screen "Automatski" 800x480
   TextField "Text field_2" at 681,0 size 116x23; Text 'Alen Lacković'
   Switch "Switch_1" at 95,185 size 160x80; CaptionText 'Switch'; TextOff 'OFF'; TextOn 'ON'
      ProcessValue <- "Automatsko_upravljanje_Paletizacija"
   TextField "Text field_4" at 95,155 size 121x28; Text 'Paletizacija'
   SymbolicIOField "Symbolic I/O field_1" at 40,317 size 130x50; TextOff '0'; TextOn '1'; TextList "Broj_komada_u_paleti_x-os"
      ProcessValue <- "Automatsko_upravljanje_Broj_komada_palete_x"
   SymbolicIOField "Symbolic I/O field_2" at 173,317 size 130x50; TextOff '0'; TextOn '1'; TextList "Broj_komada_u_paleti_y-os"
      ProcessValue <- "Automatsko_upravljanje_Broj_komada_palete_y"
   TextField "Text field_3" at 38,267 size 114x46; Text 'Broj komada u paleti x-os'
   TextField "Text field_5" at 173,267 size 114x46; Text 'Broj komada u paleti y-os'
   Switch "Switch_3" at 625,348 size 160x70; TextOn 'AUTOMATSKI REŽIM uključen'; CaptionText 'Switch'; TextOff 'RUČNI REŽIM uključen'
      ProcessValue <- "Automatsko_upravljanje_Automatski_režim"
   Button "Button_1" at 335,205 size 150x60; TextOff 'Pauza'
      on Release: InvertBit("Automatsko_upravljanje_Pauza")
      Appearance <- "Automatsko_upravljanje_Pauza"
   Switch "Switch_2" at 40,55 size 90x80; TextOn 'ON'; CaptionText 'Switch'; TextOff 'OFF'
      ProcessValue <- "Motor_DB_Motor_1_x-os_Uključi_motor"
   Switch "Switch_4" at 320,55 size 90x80; TextOn 'ON'; CaptionText 'Switch'; TextOff 'OFF'
      ProcessValue <- "Motor_DB_Motor_2_y-os_Uključi_motor"
   TextField "Text field_8" at 290,5 size 155x52; Text 'MOTOR 2 Y-OS GORE/DOLJE'
   TextField "Text field_9" at 10,5 size 159x52; Text 'MOTOR 1 X-OS LIJEVO/DESNO'
   Switch "Switch_5" at 565,185 size 160x80; TextOn 'ON'; CaptionText 'Switch'; TextOff 'OFF'
      ProcessValue <- "Automatsko_upravljanje_Lokalizacija_objekata"
   TextField "Text field_1" at 562,130 size 217x52; Text 'Lokalizacija objekata i sortiranje'
   Softkey "Softkey_F8" at 0,0 size 0x0; SoftkeyImage "Right_Arrow"
      on KeyDown: ActivateScreen("Ručni", 0)

screen "Ručni" 800x480
   Softkey "Softkey_F1" at 0,0 size 0x0; SoftkeyImage "Left_Arrow"
      on KeyDown: ActivateScreen("Automatski", 0)
   Softkey "Softkey_F8" at 0,0 size 0x0; SoftkeyImage "Right_Arrow"
      on KeyDown: ActivateScreen("Ručni_v2", 0)
   Button "Button_5" at 280,60 size 90x80; TextOff 'Homing'
      on Press: SetBit("Motor_DB_Motor_1_x-os_Pokreni_homing")
      on Release: ResetBit("Motor_DB_Motor_1_x-os_Pokreni_homing")
   Button "Button_6" at 480,60 size 90x80; TextOff 'Halt'
      on Press: SetBit("Motor_DB_Motor_1_x-os_Pokreni_zaustavljanje")
      on Release: ResetBit("Motor_DB_Motor_1_x-os_Pokreni_zaustavljanje")
   Button "Button_7" at 580,60 size 90x80; TextOff 'Move Absolute'
      on Press: SetBit("Motor_DB_Motor_1_x-os_Pokreni_izvršavanje_pomaka_apsolutno")
      on Release: ResetBit("Motor_DB_Motor_1_x-os_Pokreni_izvršavanje_pomaka_apsolutno")
   Button "Button_9" at 280,230 size 90x80; TextOff 'Homing'
      on Release: ResetBit("Motor_DB_Motor_2_y-os_Pokreni_homing")
      on Press: SetBit("Motor_DB_Motor_2_y-os_Pokreni_homing")
   Button "Button_10" at 480,230 size 90x80; TextOff 'Halt'
      on Release: ResetBit("Motor_DB_Motor_2_y-os_Pokreni_zaustavljanje")
      on Press: SetBit("Motor_DB_Motor_2_y-os_Pokreni_zaustavljanje")
   Button "Button_11" at 580,230 size 90x80; TextOff 'Move Absolute'
      on Release: ResetBit("Motor_DB_Motor_2_y-os_Pokreni_izvršavanje_pomaka_apsolutno")
      on Press: SetBit("Motor_DB_Motor_2_y-os_Pokreni_izvršavanje_pomaka_apsolutno")
   IOField "I/O field_1" at 580,190 size 90x40; FormatPattern s999.99
      ProcessValue <- "Motor_DB_Motor_2_y-os_Željena_pozicija"
   IOField "I/O field_2" at 580,20 size 90x40; FormatPattern s999.99
      ProcessValue <- "Motor_DB_Motor_1_x-os_Željena_pozicija"
   Button "Button_1" at 380,230 size 90x80; TextOff 'Reset'
      on Release: ResetBit("Motor_DB_Motor_2_y-os_Potvrdi_error(reset)")
      on Press: SetBit("Motor_DB_Motor_2_y-os_Potvrdi_error(reset)")
   Button "Button_2" at 380,60 size 90x80; TextOff 'Reset'
      on Release: ResetBit("Motor_DB_Motor_1_x-os_Potvrdi_error(reset)")
      on Press: SetBit("Motor_DB_Motor_1_x-os_Potvrdi_error(reset)")
   IOField "I/O field_3" at 85,250 size 90x40; FormatPattern s999.99
      ProcessValue <- "Motor_DB_Motor_2_y-os_Trenutna_pozicija"
   IOField "I/O field_4" at 85,80 size 90x40; FormatPattern s999.99
      ProcessValue <- "Motor_DB_Motor_1_x-os_Trenutna_pozicija"
   Button "Button_3" at 680,60 size 90x80; TextOff 'Move Realtive'
      on Release: ResetBit("Motor_DB_Motor_1_x-os_Pokreni_izvršavanje_pomaka_relativno")
      on Press: SetBit("Motor_DB_Motor_1_x-os_Pokreni_izvršavanje_pomaka_relativno")
   IOField "I/O field_5" at 680,20 size 90x40; FormatPattern s999.99
      ProcessValue <- "Motor_DB_Motor_1_x-os_Željeni_pomak"
   Button "Button_4" at 680,230 size 90x80; TextOff 'Move Relative'
      on Release: ResetBit("Motor_DB_Motor_2_y-os_Pokreni_izvršavanje_pomaka_relativno")
      on Press: SetBit("Motor_DB_Motor_2_y-os_Pokreni_izvršavanje_pomaka_relativno")
   IOField "I/O field_6" at 680,190 size 90x40; FormatPattern s999.99
      ProcessValue <- "Motor_DB_Motor_2_y-os_Željeni_pomak"
   TextField "Text field_1" at 0,170 size 182x29; Text 'Y-os (MOTOR 2 )'
   TextField "Text field_2" at 0,0 size 176x54; Text 'X-os (MOTOR 1)'
   TextField "Text field_4" at 0,75 size 80x42; Text 'Trenutna pozicija'
   TextField "Text field_5" at 0,245 size 80x42; Text 'Trenutna pozicija'
   Switch "Switch_1" at 180,60 size 90x80; CaptionText 'Switch'; TextOff 'OFF'; TextOn 'ON'
      ProcessValue <- "Motor_DB_Motor_1_x-os_Uključi_motor"
   Switch "Switch_2" at 180,230 size 90x80; TextOn 'ON'; CaptionText 'Switch'; TextOff 'OFF'
      ProcessValue <- "Motor_DB_Motor_2_y-os_Uključi_motor"
   Button "Button_8" at 30,343 size 120x80; TextOff 'CILINDAR'
      on Release: InvertBit("Pneumatske_komponente_Aktivacija_cilindra")
   Button "Button_12" at 345,343 size 120x80; TextOff 'HVATALJKA'
      on Release: InvertBit("Pneumatske_komponente_Aktivacija_hvataljke")
   SymbolicIOField "Symbolic I/O field_1" at 150,355 size 120x60; TextOn '1'; TextOff '0'; TextList "Stanje_cilindra"
      ProcessValue <- "Dist_ulaz5"
   SymbolicIOField "Symbolic I/O field_2" at 465,355 size 120x60; TextOn '1'; TextOff '0'; TextList "Stanje_hvataljke"
      ProcessValue <- "Dist_ulaz7"
   Switch "Switch_3" at 625,348 size 160x70; TextOn 'AUTOMATSKI REŽIM uključen'; CaptionText 'Switch'; TextOff 'RUČNI REŽIM uključen'
      ProcessValue <- "Automatsko_upravljanje_Automatski_režim"

screen "Ručni_v2" 800x480
   Softkey "Softkey_F1" at 0,0 size 0x0; SoftkeyImage "Left_Arrow"
      on KeyDown: ActivateScreen("Ručni", 0)
   Button "Button_1" at 40,230 size 120x80; TextOff 'LIJEVO'
      on Press: SetBit("Rucno_upravljanje_LIJEVO")
      on Release: ResetBit("Rucno_upravljanje_LIJEVO")
      Appearance <- "Motor_DB_Motor_1_x-os_Power_Status"
   Button "Button_2" at 320,230 size 120x80; TextOff 'DESNO'
      on Press: SetBit("Rucno_upravljanje_DESNO")
      on Release: ResetBit("Rucno_upravljanje_DESNO")
      Appearance <- "Motor_DB_Motor_1_x-os_Power_Status"
   Button "Button_3" at 180,140 size 120x80; TextOff 'GORE'
      on Press: SetBit("Rucno_upravljanje_GORE")
      on Release: ResetBit("Rucno_upravljanje_GORE")
      Appearance <- "Motor_DB_Motor_2_y-os_Power_Status"
   Button "Button_4" at 180,320 size 120x80; TextOff 'DOLJE'
      on Press: SetBit("Rucno_upravljanje_DOLJE")
      on Release: ResetBit("Rucno_upravljanje_DOLJE")
      Appearance <- "Motor_DB_Motor_2_y-os_Power_Status"
   Switch "Switch_1" at 40,45 size 90x80; TextOn 'ON'; CaptionText 'Switch'; TextOff 'OFF'
      ProcessValue <- "Motor_DB_Motor_1_x-os_Uključi_motor"
   Switch "Switch_2" at 320,45 size 90x80; TextOn 'ON'; CaptionText 'Switch'; TextOff 'OFF'
      ProcessValue <- "Motor_DB_Motor_2_y-os_Uključi_motor"
   TextField "Text field_1" at 320,10 size 237x28; Text 'MOTOR 2 GORE/DOLJE'
   TextField "Text field_2" at 40,10 size 259x28; Text 'MOTOR 1 LIJEVO/DESNO'
   IOField "I/O field_1" at 410,85 size 120x40; FormatPattern s99.99
      ProcessValue <- "Rucno_upravljanje_GD_brzina"
   IOField "I/O field_2" at 130,85 size 120x40; FormatPattern s99.99
      ProcessValue <- "Rucno_upravljanje_LD_brzina"
   Button "Button_5" at 510,140 size 120x80; TextOff 'CILINDAR'
      on Release: InvertBit("Pneumatske_komponente_Aktivacija_cilindra")
   Button "Button_6" at 650,140 size 120x80; TextOff 'HVATALJKA'
      on Release: InvertBit("Pneumatske_komponente_Aktivacija_hvataljke")
   SymbolicIOField "Symbolic I/O field_1" at 510,220 size 120x60; TextOff '0'; TextOn '1'; TextList "Stanje_cilindra"
      ProcessValue <- "Dist_ulaz5"
   SymbolicIOField "Symbolic I/O field_2" at 650,220 size 120x60; TextOn '1'; TextOff '0'; TextList "Stanje_hvataljke"
      ProcessValue <- "Dist_ulaz7"
   TextField "Text field_3" at 410,40 size 166x42; Text 'Unos željene brzine kretanja (30 mm/s)'
   TextField "Text field_4" at 130,40 size 166x42; Text 'Unos željene brzine kretanja (30 mm/s)'
   Switch "Switch_4" at 625,348 size 160x70; TextOn 'AUTOMATSKI REŽIM uključen'; CaptionText 'Switch'; TextOff 'RUČNI REŽIM uključen'
      ProcessValue <- "Automatsko_upravljanje_Automatski_režim"
*)